(* IEC 61131-3 sources: ICSML/Codesys_V3/Function Blocks/Input.pou, 1 file *)

(* ---- Input.pou ---- *)
(*#-#-#-#-#-#-#-#-#-#---Declaration---#-#-#-#-#-#-#-#-#-#-#-#-#*)

FUNCTION_BLOCK Input IMPLEMENTS Layer
VAR
	// Input and Output dataMem variables
	input_i: dataMem;
	output_i: dataMem;
END_VAR

(*#-#-#-#-#-#-#-#-#-#---Implementation---#-#-#-#-#-#-#-#-#-#-#-#-#*)
